PROGRAM OVERVIEW_FBD
VAR
	fbButtonBox: FB_ButtonBox;
	fbBeltControl: FB_BeltControl;
	fbGatoPerro: FB_GatoPerro;
END_VAR

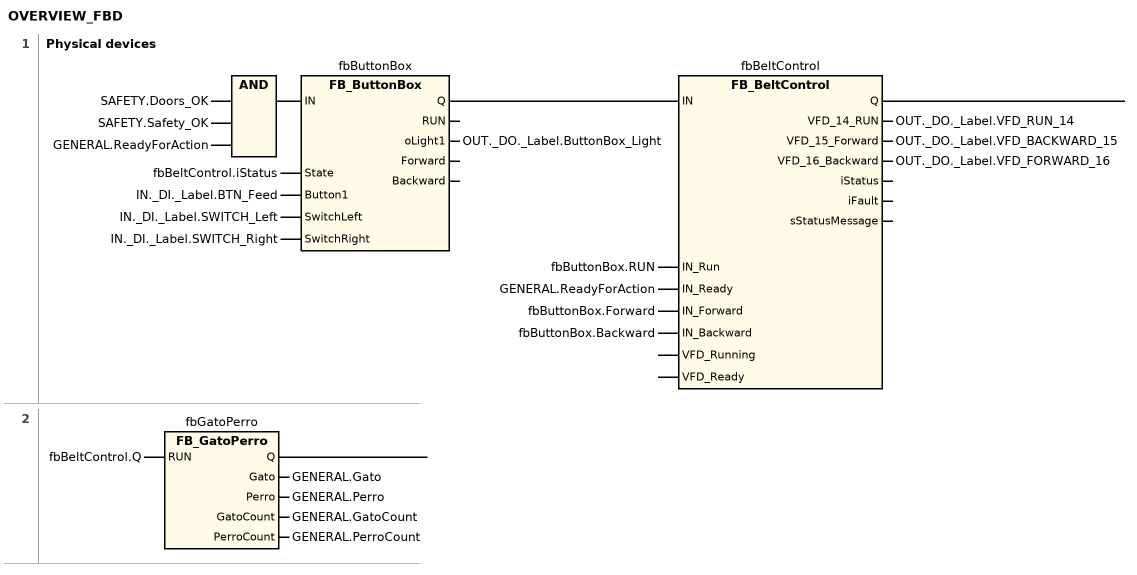
// NETWORK 1: Physical devices
fbButtonBox(
    IN := SAFETY.Doors_OK AND SAFETY.Safety_OK AND GENERAL.ReadyForAction,
    State := fbBeltControl.iStatus,
    Button1 := IN._DI._Label.BTN_Feed,
    SwitchLeft := IN._DI._Label.SWITCH_Left,
    SwitchRight := IN._DI._Label.SWITCH_Right,
    oLight1 => OUT._DO._Label.ButtonBox_Light); // FB_ButtonBox
fbBeltControl(
    IN := fbButtonBox.Q,
    IN_Run := fbButtonBox.RUN,
    IN_Ready := GENERAL.ReadyForAction,
    IN_Forward := fbButtonBox.Forward,
    IN_Backward := fbButtonBox.Backward,
    VFD_14_RUN => OUT._DO._Label.VFD_RUN_14,
    VFD_15_Forward => OUT._DO._Label.VFD_BACKWARD_15,
    VFD_16_Backward => OUT._DO._Label.VFD_FORWARD_16); // FB_BeltControl

// NETWORK 2
fbGatoPerro(
    RUN := fbBeltControl.Q,
    Gato => GENERAL.Gato,
    Perro => GENERAL.Perro,
    GatoCount => GENERAL.GatoCount,
    PerroCount => GENERAL.PerroCount); // FB_GatoPerro

END_PROGRAM

(* stored: Version 1.1.0.1, ProductVersion 3.1.4024.10
   POU OVERVIEW_FBD: Id {5015793d-548e-4713-ad62-be76714ca000}, SpecialFunc None *)
